{attribute 'linkalways'} 
{attribute 'no_explicit_call' := 'This FB is a CLASS and must be accessed using methods or properties'}
{attribute 'enable_dynamic_creation'}
{attribute 'hide_all_locals'}
FUNCTION_BLOCK Extension EXTENDS Disposable IMPLEMENTS I_Extension
VAR
	_name : T_MAXSTRING;
	_parent : I_HostExtensions;
	eventEmitter : EventEmitter;
	inputPortHost : InputPortHost(THIS^, eventEmitter);
	outputPortHost : OutputPortHost(THIS^, eventEmitter);
	parameterHost : ParameterHost(THIS^, eventEmitter);
	contentHost : ContentHost(THIS^, eventEmitter);
	alarmHost : AlarmHost(THIS^, eventEmitter);
	metadataHost : MetadataHost(THIS^, eventEmitter);
	deserializationFailedAlarm : DeserializationFailedAlarm(THIS^);
END_VAR

METHOD PUBLIC Accept
VAR_INPUT
	Visitor : I_ExtensionVisitor;
END_VAR
Visitor.VisitExtension(THIS^);
END_METHOD

METHOD PROTECTED AddContent : I_Content
VAR_INPUT
	Name : T_MAXSTRING;
	Data : I_Datatype;
END_VAR
AddContent := Contents.AddDataAsContent(Name, Data);
END_METHOD

METHOD PROTECTED AddInput : I_InputPort
VAR_INPUT
	Name : T_MAXSTRING;
	Data : I_Datatype;
END_VAR
AddInput := InputPorts.AddDataAsInputPort(Name, Data);
END_METHOD

METHOD PUBLIC AddMetadata : I_HostMetadata
VAR_INPUT
	Name : T_MAXSTRING;
	Data : I_Datatype;
END_VAR
Metadatum.AddDataAsMetadata(Name, Data);
AddMetadata := THIS^;
END_METHOD

METHOD PROTECTED AddOutput : I_OutputPort
VAR_INPUT
	Name : T_MAXSTRING;
	Data : I_Datatype;
END_VAR
AddOutput := OutputPorts.AddDataAsOutputPort(Name, Data);
END_METHOD

METHOD PROTECTED AddParameter : I_Parameter
VAR_INPUT
	Name : T_MAXSTRING;
	Data : I_Datatype;
END_VAR
AddParameter := Parameters.AddDataAsParameter(Name, Data);
END_METHOD

PROPERTY PUBLIC Alarms : I_Alarms
GET
Alarms := alarmHost;
END_GET
END_PROPERTY

PROPERTY PUBLIC Contents : I_Contents
GET
Contents := contentHost;
END_GET
END_PROPERTY

METHOD FB_init : BOOL
VAR_INPUT
	bInitRetains : BOOL; // if TRUE, the retain variables are initialized (warm start / cold start)
	bInCopyCode : BOOL;  // if TRUE, the instance afterwards gets moved into the copy code (online change)
	Name : T_MAXSTRING;
	Parent : I_HostExtensions;
END_VAR
_name := Name;
RegisterWithParent(Parent);
END_METHOD

PROPERTY PUBLIC HasRaisedAlarm : BOOL
GET
HasRaisedAlarm := alarmHost.HasRaisedAlarm;
END_GET
END_PROPERTY

PROPERTY PUBLIC InputPorts : I_InputPorts
GET
InputPorts := inputPortHost;
END_GET
END_PROPERTY

PROPERTY PUBLIC Metadatum : I_Metadatum
GET
Metadatum := metadataHost;
END_GET
END_PROPERTY

PROPERTY PUBLIC Name : T_MAXSTRING
GET
Name := _name;
END_GET
END_PROPERTY

METHOD PUBLIC OffEvent
VAR_INPUT
	EventName : T_MaxString;
	EventHandler : I_EventHandler;
END_VAR
eventEmitter.OffEvent(EventName, EventHandler);
END_METHOD

METHOD PUBLIC OnceEvent
VAR_INPUT
	EventName : T_MaxString;
	EventHandler : I_EventHandler;
END_VAR
eventEmitter.OnceEvent(EventName, EventHandler);
END_METHOD

METHOD PUBLIC OnEvent
VAR_INPUT
	EventName : T_MaxString;
	EventHandler : I_EventHandler;
END_VAR
eventEmitter.OnEvent(EventName, EventHandler);
END_METHOD

PROPERTY PUBLIC OutputPorts : I_OutputPorts
GET
OutputPorts := outputPortHost;
END_GET
END_PROPERTY

PROPERTY PUBLIC Parameters : I_Parameters
GET
Parameters := parameterHost;
END_GET
END_PROPERTY

PROPERTY PUBLIC Parent : I_HostExtensions
GET
Parent := _parent;
END_GET
END_PROPERTY

METHOD PUBLIC RegisterWithParent
VAR_INPUT
	Parent : I_HostExtensions;
END_VAR
IF Parent = 0 THEN
	RETURN;
END_IF

_parent := Parent;
Parent.Extensions.AddExtension(THIS^);
END_METHOD

METHOD PUBLIC SerializeWith
VAR_INPUT
	Serializer : I_Serializer;
END_VAR
Serializer.StartObject();
Serializer.AddKeyString('name', _name);
inputPortHost.SerializeWith(Serializer);
outputPortHost.SerializeWith(Serializer);
parameterHost.SerializeWith(Serializer);
contentHost.SerializeWith(Serializer);
alarmHost.SerializeWith(Serializer);
metadataHost.SerializeWith(Serializer);
Serializer.EndObject();
END_METHOD

METHOD PUBLIC TryDeserializeFrom : BOOL
VAR_INPUT
	Deserializer : I_Deserializer;
	Feedback : I_DeserializerFeedback;
END_VAR
DeserializationFailedAlarm.Clear();

IF NOT parameterHost.TryDeserializeFrom(Deserializer, Feedback) THEN
	DeserializationFailedAlarm.Raise('Failed to deserialize parameters');
	RETURN;
END_IF

TryDeserializeFrom := TRUE;
END_METHOD

END_FUNCTION_BLOCK

(* stored: Version 1.1.0.1, ProductVersion 3.1.4024.13
   POU Extension: Id {8ac7b2c9-5c38-4780-b32e-134f1c230d16}, SpecialFunc None
   Folder Constructor: Id {e2fa132a-df47-4d80-943f-0757a42d94ae}
   Folder Protected: Id {600cde5a-f526-03d2-1972-8f756ca519e8}
   Method Accept: Id {c2d85c76-9431-4c14-8ff5-79e11f782333}
   Method AddContent: Id {0f917303-57db-0e31-09c9-7ec26ec41fe1}
   Method AddInput: Id {2581c864-368b-062b-2420-fc4a344b3c81}
   Method AddMetadata: Id {f2addbcd-14f3-0a89-15e5-56d36063222e}
   Method AddOutput: Id {8d942aae-84b8-0551-371a-141e14b70a72}
   Method AddParameter: Id {fbb602a7-dd34-0193-1623-f33becde78d3}
   Property Alarms: Id {7a9d58bb-1bd2-477c-8b87-11fa3ac91181}
   Get Get: Id {e2e4c3c0-367e-4f2c-93d3-b034a6193124}
   Property Contents: Id {d4deca99-c794-4842-9f14-2120be9cdc35}
   Get Get: Id {6b8cac52-6ee9-48c0-b6d7-deb24e0974c5}
   Method FB_init: Id {194b9380-c1ce-437f-9678-bce9e9aee887}
   Property HasRaisedAlarm: Id {4c3dd4a1-3f0e-441e-a770-d854acec24f5}
   Get Get: Id {d127264d-ae92-4a8e-b80e-ba8b6a9d61df}
   Property InputPorts: Id {3e312d95-ab25-4eca-af6a-c42cecf8b452}
   Get Get: Id {db14c4a7-51cc-493f-872c-cdc8a77f85bc}
   Property Metadatum: Id {eab8e526-6a6c-4991-bdcf-4229c8e8a72b}
   Get Get: Id {c1bfc407-406b-4ae3-805d-fffc431f10cc}
   Property Name: Id {c85fa46e-ae0e-48b2-be11-4ec1413abe4e}
   Get Get: Id {b20c0a68-16b8-4d8a-ae96-15a0b0d9c536}
   Method OffEvent: Id {6835458e-f377-4a82-8de0-709c8a6186bb}
   Method OnceEvent: Id {12d2564f-8b36-4596-8526-8ba3d0358ff0}
   Method OnEvent: Id {e99a5517-2019-486d-8aee-8229c32d654c}
   Property OutputPorts: Id {2185d460-f262-46ff-a85e-79554489b2d3}
   Get Get: Id {03e5674a-3fff-4e57-bf57-4fb7138aaabf}
   Property Parameters: Id {a78eeb0a-232e-4885-afc3-eea8a907e31d}
   Get Get: Id {c460ccdb-7185-41a6-8d7c-02e232aa6cf2}
   Property Parent: Id {c55a2944-e008-06dc-1879-15847c089e2e}
   Get Get: Id {4f3f87b8-092f-0670-104f-8505892f987f}
   Method RegisterWithParent: Id {b5b82bae-9e1c-0474-17d5-193b4bb784ed}
   Method SerializeWith: Id {6685483b-02aa-44da-bca9-467fc317fca6}
   Method TryDeserializeFrom: Id {f1cd085b-4b54-41dd-a2be-f0cb8ced9794} *)
